// TIA Portal V18 export
DATA_BLOCK "IAI_DeviceCtl"   // DB2204
{ S7_Optimized_Access := 'FALSE' }
VERSION : 0.1
// stored: AutoNumber false, DBAccessibleFromOPCUA true, DBAccessibleFromWebserver true, IsOnlyStoredInLoadMemory false, IsWriteProtectedInAS false
   VAR RETAIN
      IAIServo : Array[1..4] of Struct
         i : Int;
         nError : Int;
         nWarning : Int;
         nPositionListNo : Int;
         Pos : "PosList_IAI";
         Point : Array[0..39] of Struct
            Start : Bool;
            Achieve : Bool;
         END_STRUCT;
      END_STRUCT;
   END_VAR
BEGIN
   IAIServo[1..4].nPositionListNo := 1;
   // IAIServo[1].Point[1] : 初始位 / 上料位1
   // IAIServo[1].Point[2] : 抓料位 / 上料位2
   // IAIServo[1].Point[3] : 上料拍照位 / 上料位3
   // IAIServo[1].Point[4] : 下料位1 / 上料位4
   // IAIServo[1].Point[5] : 下料位2 / 上料位5
   // IAIServo[1].Point[6] : 下料位3 / 上料位6
   // IAIServo[1].Point[7] : 下料位4 / 上料位7
   // IAIServo[1].Point[8] : 下料位5 / 上料位8
   // IAIServo[1].Point[9] : NG下料位
   // IAIServo[2].Point[1] : 初始位
   // IAIServo[2].Point[2] : 取料位1 / 扫码位置2
   // IAIServo[2].Point[3] : 取料位2 / 扫码位置3
   // IAIServo[2].Point[4] : 取料位3 / 扫码位置4
   // IAIServo[2].Point[5] : 取料位4 / 扫码位置5
   // IAIServo[2].Point[6] : 取料位5 / 扫码位置6
   // IAIServo[2].Point[7] : 清洁位 / 扫码位置7
   // IAIServo[2].Point[8] : NG位 / 扫码位置8
   // IAIServo[2].Point[9] : 快速装配位
   // IAIServo[2].Point[10] : 慢速装配位
END_DATA_BLOCK
